TYPE "MEStoPLC_ProcessingExchange"
VERSION : 0.1
   STRUCT
      "M-ProcessingDone" : Bool;
      Reserve : Array[1..298] of Byte;
   END_STRUCT;

END_TYPE

